FUNCTION_BLOCK STEPPER (* Basic Function Block Type *)
  (* Standard: 61499-2 *)
  (* Version 0.0, 4/28/2023, Dmitrii, Flexbridge AB, Template *)
  PACKAGE UAO.Hackathon;
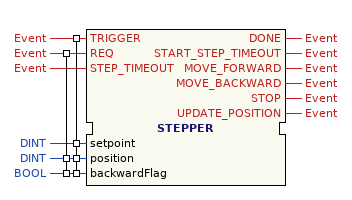
  EVENT_INPUT
    TRIGGER WITH position, setpoint, backwardFlag; (* Start stepping towards the setpoint *)
    REQ WITH position, backwardFlag; (* Update values *)
    STEP_TIMEOUT;
  END_EVENT
  EVENT_OUTPUT
    DONE; (* Movement complete *)
    START_STEP_TIMEOUT;
    MOVE_FORWARD;
    MOVE_BACKWARD;
    STOP;
    UPDATE_POSITION;
  END_EVENT
  VAR_INPUT
    setpoint : DINT; (* Target position *)
    position : DINT; (* current position *)
    backwardFlag : BOOL;
  END_VAR
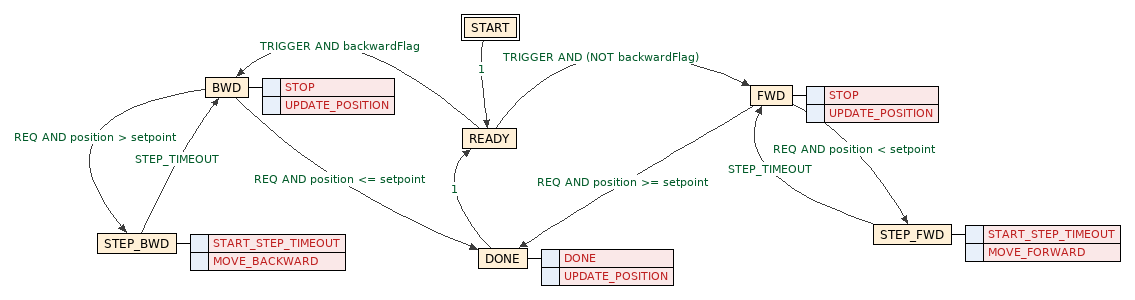
  EC_STATES
    START; (* Initial State *)
    READY;
    FWD : -> STOP, -> UPDATE_POSITION;
    STEP_FWD : -> START_STEP_TIMEOUT, -> MOVE_FORWARD;
    DONE : -> DONE, -> UPDATE_POSITION;
    BWD : -> STOP, -> UPDATE_POSITION;
    STEP_BWD : -> START_STEP_TIMEOUT, -> MOVE_BACKWARD;
  END_STATES
  EC_TRANSITIONS
    START TO READY := 1;
    FWD TO STEP_FWD := REQ AND position < setpoint;
    STEP_FWD TO FWD := STEP_TIMEOUT;
    DONE TO READY := 1;
    FWD TO DONE := REQ AND position >= setpoint;
    READY TO FWD := TRIGGER AND (NOT backwardFlag);
    READY TO BWD := TRIGGER AND backwardFlag;
    BWD TO STEP_BWD := REQ AND position > setpoint;
    STEP_BWD TO BWD := STEP_TIMEOUT;
    BWD TO DONE := REQ AND position <= setpoint;
  END_TRANSITIONS
  ALGORITHM INIT IN ST: (* Initialization algorithm *)
;
  END_ALGORITHM
END_FUNCTION_BLOCK
